(* CODESYS project PLS2 Trykkregulering 19.07.2021.ecp

Project tree, tasks and I/O mapping:
  PFCx00_SmartCoupler : 750-8212 PFC200 2ETH RS, WAGO, order no. 0750-8212, version 5.15.4.20
    application PLS2_Trykkregulering
      libraries: ; VisuDialogs, * (System); WagoTypesCommon, 1.5.3.0 (WAGO); WagoAppHART, 1.7.1.0 (WAGO); WagoAppSolenoid, 1.7.1.0 (WAGO); WagoAppPowerMeasurement, 1.7.1.0 (WAGO); WagoTypesCom, 1.6.1.2 (WAGO); WagoAppDALI, 1.3.0.33 (WAGO); WagoSysKbusModule, 1.8.2.0 (WAGO); WagoSysKbusServices, 1.8.7.4 (WAGO); WagoAppPlcModbus, 1.1.2.21 (WAGO); WagoTypesAsync_Internal_Template, 1.0.0.1 (WAGO); WagoSysModule_75x_632, 1.8.1.0 (WAGO); WagoSysModule_75x_48x, 1.5.1.0 (WAGO); WagoVisuIcons, 1.0.1.0 (WAGO); WagoSysModule_75x_49x, 1.7.1.0 (WAGO); WagoSysModule_753_647, 1.1.1.0 (WAGO); WagoAppKNX, 1.0.4.0 (WAGO); WagoAppCloud, * (WAGO); WagoAppTime, 1.7.3.3 (WAGO); WagoAppJSON, 1.0.2.0 (WAGO); CmpEventMgr, 3.5.12.0 (System); Component Manager, 3.5.13.0 (System); CmpApp, 3.5.13.0 (System); CmpIecTask, 3.5.13.0 (System)
      task PLC_Task (cyclic, interval 100 ms, priority 10, watchdog 90 ms x 1) calls PLC_PRG
      task VISU_TASK (cyclic, interval 100 ms, priority 15) calls VisuElems.Visu_Prg
      task TrendRecordingTask (cyclic, interval 100 ms, priority 15) calls VisuTrendStorageAccess.GlobalInstances.g_TrendRecordingManager.CyclicCall
      program PLC_PRG [ST]
      program Alarms [ST]
      GlobalData/
        global variables HMI
        global variables Local
        global variables IO
        global variables SIM
        global variables STATUS
      Symbols
      program Inputs [ST]
      program Control [ST]
      program Outputs [ST]
      program Simulation [ST]
      program Initialize [ST]
      visualisation Visualization
      global variables PersistentVars
      function RestartOpcUaMqttLinkOnDownload [ST]
      function RestartOpcUaMqttLinkOnOnlineChange [ST]
    ProjectConfigurationTxt
    ProjectConfiguration
    Common.PCI
    Kbus : Kbus, WAGO, version 1.4.0.2
        unmapped channels: K-BUS diagnostics
    MODBUS
      MODBUS : MODBUS, WAGO, order no. n/a, version 1.1.1.15
    Serial
      COM1 : COM1, WAGO, version 0.0.0.19
  00000000-0000-0000-0000-000000000000|C:\Users\WagoNorgeLab-1\AppData\Local\Temp\ee55296a4ebe4169b370fb7549785af2\ProjectCfg.txt
  LibFB/
    function block AlarmDigitalFB [ST]
    function block MotorDigitalFB [ST]
    function block ControlAnalogFB [ST]
    function block ScalingFB [ST]
    function block signalDigitalFB [ST]
    function block TimerFB [ST]
    function block SignalAnalogFB [ST]
    function block PIDFB [ST]
    function block WorkDistributorFB [ST]
  LibHmiStructs/
    data type AlarmDigitalHmiPv
    data type ControlAnalogHmiPv
    data type MotorDigitalHmiPv
    data type MotorDigitalHmiCmd
    data type ControlAnalogHmiCmd
    data type AlarmDigitalHmiCmd
    data type TimerHmiPv
    data type TimerHmiCmd
    data type SignalDigitalHmiPv
    data type SignalDigitalHmiCmd
    data type ScalingHmiPv
    data type ScalingHmiCmd
    data type SignalAnalogHmiPv
    data type SignalAnalogHmiCmd
    data type AliveHmiPv
    data type PIDHmiCmd
    data type PIDHmiPv
    data type WorkDistributorHmiPv
  Utils/
    function eulers [ST]
    function process [ST]
    function String_To_ForcastArray [ST]
    data type OpcUa_Mqtt_Status
    function firstOrderSystem [ST]
  text list GlobalTextList
  00000000-0000-0000-0000-000000000000|C:\Users\WagoNorgeLab-1\AppData\Local\Temp\0890fa1c76c045128ce9e2a1421b24b3\Project.xml
*)

// LibHmiStructs/AlarmDigitalHmiPv
// These are autogenerated, do not manual modify it
TYPE AlarmDigitalHmiPv :
STRUCT
	_tagId: STRING;
	_type: STRING;
	_owner: STRING;
	Input_Pv:	BOOL;
	Delay:	TimerHmiPv;
	Alarm:	BOOL;
END_STRUCT
END_TYPE

// LibHmiStructs/ControlAnalogHmiPv
// These are autogenerated, do not manual modify it
TYPE ControlAnalogHmiPv :
STRUCT
	_tagId: STRING;
	_type: STRING;
	_owner: STRING;
	ControlValue_Pv:	REAL;
	Interlocked_Pv:	BOOL;
	AlarmControlFailed:	AlarmDigitalHmiPv;
	Feedback_Pv:REAL;
	RunHours_Pv:INT;
	RunMinutes_Pv:int;
END_STRUCT
END_TYPE

// LibHmiStructs/MotorDigitalHmiPv
// These are autogenerated, do not manual modify it
TYPE MotorDigitalHmiPv :
STRUCT
_tagId: STRING;
_type: STRING;
_owner: STRING;
Interlocked_Pv:BOOL;
ControlValue_Pv:BOOL;
AlarmStartFailed:AlarmDigitalHmiPv;
AlarmStopFailed:AlarmDigitalHmiPv;
Started_Pv:BOOL;
Stopped_Pv:BOOL;
END_STRUCT
END_TYPE

// LibHmiStructs/MotorDigitalHmiCmd
// These are autogenerated, do not manual modify it
TYPE MotorDigitalHmiCmd :
STRUCT
_tagId: STRING;
_type: STRING;
_owner: STRING;
Tag:STRING;
Description:STRING;
Auto:BOOL;
AlarmStartFailed:AlarmDigitalHmiCmd;
AlarmStopFailed:AlarmDigitalHmiCmd;
ManualStart_Cmd:BOOL;
END_STRUCT
END_TYPE

// LibHmiStructs/ControlAnalogHmiCmd
// These are autogenerated, do not manual modify it
TYPE ControlAnalogHmiCmd :
STRUCT
	_tagId: STRING;
	_type: STRING;
	_owner: STRING;
	Tag:STRING;
	Description:STRING;
	Auto:BOOL;
	ManualControlValue_Cmd:REAL;
	AlarmControlFailed:	AlarmDigitalHmiCmd;
	AlarmControlFailedLimit:	REAL;
END_STRUCT
END_TYPE

// LibHmiStructs/AlarmDigitalHmiCmd
// These are autogenerated, do not manual modify it
TYPE AlarmDigitalHmiCmd :
STRUCT
	_tagId: STRING;
	_type: STRING;
	_owner: STRING;
	Tag:	STRING;
	Description:	STRING;
	Delay:	TimerHmiCmd;
	Acknowledged:	BOOL;
END_STRUCT
END_TYPE

// LibHmiStructs/TimerHmiPv
// These are autogenerated, do not manual modify it
TYPE TimerHmiPv :
STRUCT
	_tagId:STRING;
	_type: STRING;
	_owner: STRING;
	Input_Pv:	BOOL;
	Output_Pv:	BOOL;
	OnDelayElapsed:	REAL;
	OffDelayElapsed:	REAL;
END_STRUCT
END_TYPE

// LibHmiStructs/TimerHmiCmd
// These are autogenerated, do not manual modify it
TYPE TimerHmiCmd :
STRUCT
	_tagId:STRING;
	_type: STRING;
	_owner: STRING;
	Tag:	STRING;
	Description:	STRING;
	OnDelayLimit:	REAL;
	OffDelayLimit:	REAL;
END_STRUCT
END_TYPE

// LibHmiStructs/SignalDigitalHmiPv
// These are autogenerated, do not manual modify it
TYPE SignalDigitalHmiPv :
STRUCT
_tagId: STRING;
_type: STRING;
_owner: STRING;
Input_Pv:BOOL;
Output_Pv:BOOL;
END_STRUCT
END_TYPE

// LibHmiStructs/SignalDigitalHmiCmd
// These are autogenerated, do not manual modify it
TYPE SignalDigitalHmiCmd :
STRUCT
_tagId: STRING;
_type: STRING;
_owner: STRING;
Tag:STRING;
Description:STRING;
SimulationMode:BOOL;
SimulationValue:BOOL;
END_STRUCT
END_TYPE

// LibHmiStructs/ScalingHmiPv
// These are autogenerated, do not manual modify it
TYPE ScalingHmiPv :
STRUCT
_tagId: STRING;
_type: STRING;
_owner: STRING;
Input_Pv:REAL;
Output_Pv:REAL;
END_STRUCT
END_TYPE

// LibHmiStructs/ScalingHmiCmd
// These are autogenerated, do not manual modify it
TYPE ScalingHmiCmd :
STRUCT
	_tagId: STRING;
	_type: STRING;
	_owner: STRING;
	InputUnit:STRING;
	InputMin_Cmd:REAL;
	InputMax_Cmd:REAL;
	OutputUnit:STRING;
	OutputMin_Cmd:REAL;
	OutputMax_Cmd:REAL;
END_STRUCT
END_TYPE

// LibHmiStructs/SignalAnalogHmiPv
// These are autogenerated, do not manual modify it
TYPE SignalAnalogHmiPv :
STRUCT
_tagId: STRING;
_type: STRING;
_owner: STRING;
RawInput_Pv:REAL;
Output_Pv:REAL;
AlarmHigh:AlarmDigitalHmiPv;
AlarmHighHigh:AlarmDigitalHmiPv;
AlarmLow:AlarmDigitalHmiPv;
AlarmLowLow:AlarmDigitalHmiPv;
InputScaling:ScalingHmiPv;
END_STRUCT
END_TYPE

// LibHmiStructs/SignalAnalogHmiCmd
// These are autogenerated, do not manual modify it
TYPE SignalAnalogHmiCmd :
STRUCT
_tagId: STRING;
_type: STRING;
_owner: STRING;
Tag:STRING;
Description:STRING;
AlarmHigh:AlarmDigitalHmiCmd;
AlarmHighHigh:AlarmDigitalHmiCmd;
AlarmLow:AlarmDigitalHmiCmd;
AlarmLowLow:AlarmDigitalHmiCmd;
AlarmHighLimit:REAL;
AlarmHighHighLimit:REAL;
AlarmLowLimit:REAL;
AlarmLowLowLimit:REAL;
AlarmHysteresis:REAL;
SimulationMode:BOOL;
SimulationValue:REAL;
InputScaling:ScalingHmiCmd;
END_STRUCT
END_TYPE

// LibHmiStructs/AliveHmiPv
TYPE AliveHmiPv :
STRUCT
	_tagId:STRING;
	_type: STRING;
	_owner: STRING;
	CounterPv:INT;
END_STRUCT
END_TYPE

// LibHmiStructs/PIDHmiCmd
TYPE PIDHmiCmd :
STRUCT
	_tagId: STRING;
	_type: STRING;
	_owner: STRING;
	Tag:STRING;
	Description:STRING;
	K:REAL;
	EnableK:BOOL;
	Ti:REAL;
	EnableI:BOOL;
	Td:REAL;
	N:REAL;
	EnableD:BOOL;
	Auto:BOOL;
	ManualValue_Cmd:REAL;
	u0:REAL;
	TrackingGain:REAL;
	HmiReference_Cmd:REAL;
	HmiReference:BOOL;
END_STRUCT
END_TYPE

// LibHmiStructs/PIDHmiPv
TYPE PIDHmiPv :
STRUCT
	_tagId: STRING;
	_type: STRING;
	_owner: STRING;
	Reference_Pv:REAL;
	ProcessMeasure:REAL;
	Error:REAL;
	Output:REAL;
	up:REAL;
	ui:REAL;
	ud:REAL;
	es:REAL;
	u:REAL;
END_STRUCT
END_TYPE

// Utils/OpcUa_Mqtt_Status
TYPE OpcUa_Mqtt_Status :
STRUCT
	LastRun:STRING;
	AliveCounterPv:INT := 0;
	Restart_Cmd:BOOL := FALSE;
END_STRUCT
END_TYPE

// LibHmiStructs/WorkDistributorHmiPv
TYPE WorkDistributorHmiPv :
STRUCT
_tagId:STRING;
_type:STRING;
_owner:STRING;
Tag1:STRING;
Tag2:STRING;
Tag3:STRING;
RunHours1:INT;
RunHours2:INT;
RunHours3:INT;
AlarmNotAuto:BOOL;
END_STRUCT
END_TYPE

// PFCx00_SmartCoupler/PLS2_Trykkregulering/GlobalData/HMI
{attribute 'qualified_only'}
VAR_GLOBAL PERSISTENT RETAIN
AliveCounterPlc2Pv:AliveHmiPv;

DeliveryPump1Cmd:ControlAnalogHmiCmd;
DeliveryPump1Pv:ControlAnalogHmiPv;
DeliveryPump2Cmd:ControlAnalogHmiCmd;
DeliveryPump2Pv:ControlAnalogHmiPv;
DeliveryPump3Cmd:ControlAnalogHmiCmd;
DeliveryPump3Pv:ControlAnalogHmiPv;
DeliveryPumpPIDCmd:PIDHmiCmd;
DeliveryPumpPIDPv:PIDHmiPv;
DeliveryPumpWorkDistPv:WorkDistributorHmiPv;
TreatmentPressureCmd:SignalAnalogHmiCmd;
TreatmentPressurePv:SignalAnalogHmiPv;
ConsumerPressureCmd:SignalAnalogHmiCmd;
ConsumerPressurePv:SignalAnalogHmiPv;
END_VAR

// PFCx00_SmartCoupler/PLS2_Trykkregulering/GlobalData/Local
{attribute 'qualified_only'}
VAR_GLOBAL
DeliveryPump1:ControlAnalogFB;
DeliveryPump2:ControlAnalogFB;
DeliveryPump3:ControlAnalogFB;
DeliveryPumpPID:PIDFB;
DeliveryPumpWorkDist:WorkDistributorFB;
TreatmentPressure:SignalAnalogFB;
ConsumerPressure:SignalAnalogFB;
END_VAR

// PFCx00_SmartCoupler/PLS2_Trykkregulering/GlobalData/IO
{attribute 'qualified_only'}
VAR_GLOBAL
AI_DeliveryPump1SpeedPv:REAL;
AI_DeliveryPump2SpeedPv:Real;
AI_DeliveryPump3SpeedPv:Real;

AO_DeliveryPump1ControlValue:real;
AO_DeliveryPump2ControlValue:real;
AO_DeliveryPump3ControlValue:REAL;

AI_ConsumerPressurePv:REAL;
AI_TreatmentPressurePv:REAL;
END_VAR

// PFCx00_SmartCoupler/PLS2_Trykkregulering/GlobalData/SIM
{attribute 'qualified_only'}
VAR_GLOBAL
	Disturbance:REAL;
	Process_y:REAL;
	Process:REAL;
	Ref:REAL;
	Output:REAL;
END_VAR

// PFCx00_SmartCoupler/PLS2_Trykkregulering/GlobalData/STATUS
{attribute 'qualified_only'}
VAR_GLOBAL
	OpcUaMqttLinkStatus: OpcUa_Mqtt_Status;
END_VAR

// PFCx00_SmartCoupler/PLS2_Trykkregulering/PersistentVars
{attribute 'qualified_only'}
VAR_GLOBAL PERSISTENT RETAIN
	// Generated instance path of persistent variable
	HMI.AliveCounterPlc2Pv: AliveHmiPv;
	// Generated instance path of persistent variable
	HMI.DeliveryPump1Cmd: ControlAnalogHmiCmd;
	// Generated instance path of persistent variable
	HMI.DeliveryPump1Pv: ControlAnalogHmiPv;
	// Generated instance path of persistent variable
	HMI.DeliveryPump2Cmd: ControlAnalogHmiCmd;
	// Generated instance path of persistent variable
	HMI.DeliveryPump2Pv: ControlAnalogHmiPv;
	// Generated instance path of persistent variable
	HMI.DeliveryPump3Cmd: ControlAnalogHmiCmd;
	// Generated instance path of persistent variable
	HMI.DeliveryPump3Pv: ControlAnalogHmiPv;
	// Generated instance path of persistent variable
	HMI.DeliveryPumpPIDCmd: PIDHmiCmd;
	// Generated instance path of persistent variable
	HMI.DeliveryPumpPIDPv: PIDHmiPv;
	// Generated instance path of persistent variable
	HMI.DeliveryPumpWorkDistPv: WorkDistributorHmiPv;
	// Generated instance path of persistent variable
	HMI.TreatmentPressureCmd: SignalAnalogHmiCmd;
	// Generated instance path of persistent variable
	HMI.TreatmentPressurePv: SignalAnalogHmiPv;
	// Generated instance path of persistent variable
	HMI.ConsumerPressureCmd: SignalAnalogHmiCmd;
	// Generated instance path of persistent variable
	HMI.ConsumerPressurePv: SignalAnalogHmiPv;
END_VAR

// PFCx00_SmartCoupler/PLS2_Trykkregulering/PLC_PRG
PROGRAM PLC_PRG
VAR
	_firstScan:BOOL := TRUE;
	_counter:INT;
	_lastRun:STRING;
END_VAR



// Signaling that the PLC is alive
Hmi.AliveCounterPlc2Pv._tagId := 'AliveCounterPlc2Pv';
Hmi.AliveCounterPlc2Pv._type := 'AliveHmi';
Hmi.AliveCounterPlc2Pv._owner := 'plc2';
HMI.AliveCounterPlc2Pv.CounterPv := HMI.AliveCounterPlc2Pv.CounterPv + 1;

_counter := STATUS.OpcUaMqttLinkStatus.AliveCounterPv;
_lastRun := STATUS.OpcUaMqttLinkStatus.LastRun;

IF _firstScan THEN
	Initialize();
END_IF
Inputs();
Alarms();
Control();
Outputs();
Simulation();





// Always last
_firstScan := FALSE;

END_PROGRAM

// PFCx00_SmartCoupler/PLS2_Trykkregulering/Initialize
PROGRAM Initialize
VAR
END_VAR



Hmi.DeliveryPumpPIDCmd.Tag := 'PID01';
Hmi.DeliveryPumpPIDCmd.Description := 'Regulator for controling pressure';
Hmi.DeliveryPumpPIDCmd.Auto := TRUE;
Hmi.DeliveryPumpPIDCmd.EnableK := TRUE;
Hmi.DeliveryPumpPIDCmd.EnableI := TRUE;
Hmi.DeliveryPumpPIDCmd.EnableD := TRUE;
Hmi.DeliveryPumpPIDCmd.K := 8.0;
Hmi.DeliveryPumpPIDCmd.Ti := 5.5;
Hmi.DeliveryPumpPIDCmd.Td := 0.5;
Hmi.DeliveryPumpPIDCmd.N := 10.0;
Hmi.DeliveryPumpPIDCmd.TrackingGain := 1.0;
Hmi.DeliveryPumpPIDCmd.u0 := 50.0;


HMI.DeliveryPump1Cmd.Tag := 'P01';
HMI.DeliveryPump1Cmd.Description := 'Delivery pump 1';
HMI.DeliveryPump1Cmd.Auto := TRUE;
HMI.DeliveryPump1Cmd.ManualControlValue_Cmd := 50.0;
HMI.DeliveryPump1Cmd.AlarmControlFailedLimit := 10.0;
HMI.DeliveryPump1Cmd.AlarmControlFailed.Description := 'Failed to control Delivery Pump 1';
HMI.DeliveryPump1Cmd.AlarmControlFailed.Delay.OnDelayLimit := 10.0;
HMI.DeliveryPump1Cmd.AlarmControlFailed.Delay.OffDelayLimit := 10.0;
HMI.DeliveryPump1Cmd.AlarmControlFailed.Acknowledged := TRUE;

HMI.DeliveryPump2Cmd.Tag := 'P02';
HMI.DeliveryPump2Cmd.Description := 'Delivery pump 2';
HMI.DeliveryPump2Cmd.Auto := TRUE;
HMI.DeliveryPump2Cmd.ManualControlValue_Cmd := 50.0;
HMI.DeliveryPump2Cmd.AlarmControlFailedLimit := 10.0;
HMI.DeliveryPump2Cmd.AlarmControlFailed.Description := 'Failed to control Delivery Pump 2';
HMI.DeliveryPump2Cmd.AlarmControlFailed.Delay.OnDelayLimit := 10.0;
HMI.DeliveryPump2Cmd.AlarmControlFailed.Delay.OffDelayLimit := 10.0;
HMI.DeliveryPump2Cmd.AlarmControlFailed.Acknowledged := TRUE;

HMI.DeliveryPump3Cmd.Tag := 'P03';
HMI.DeliveryPump3Cmd.Description := 'Delivery pump 2';
HMI.DeliveryPump3Cmd.Auto := TRUE;
HMI.DeliveryPump3Cmd.ManualControlValue_Cmd := 50.0;
HMI.DeliveryPump3Cmd.AlarmControlFailedLimit := 10.0;
HMI.DeliveryPump3Cmd.AlarmControlFailed.Description := 'Failed to control Delivery Pump 3';
HMI.DeliveryPump3Cmd.AlarmControlFailed.Delay.OnDelayLimit := 10.0;
HMI.DeliveryPump3Cmd.AlarmControlFailed.Delay.OffDelayLimit := 10.0;
HMI.DeliveryPump3Cmd.AlarmControlFailed.Acknowledged := TRUE;

Hmi.TreatmentPressureCmd.Tag := 'PT02';
Hmi.TreatmentPressureCmd.Description := 'Treatment pressure';
Hmi.TreatmentPressureCmd.AlarmHysteresis := 3.0;
Hmi.TreatmentPressureCmd.AlarmHighHighLimit := 90.0;
Hmi.TreatmentPressureCmd.AlarmHighLimit := 80.0;
Hmi.TreatmentPressureCmd.AlarmLowLowLimit := 10.0;
Hmi.TreatmentPressureCmd.AlarmLowLimit := 20.0;
Hmi.TreatmentPressureCmd.AlarmHigh.Description := 'High Treatment Pressure';
Hmi.TreatmentPressureCmd.AlarmHighHigh.Description := 'High high Treatment Pressure';
Hmi.TreatmentPressureCmd.AlarmLow.Description := 'Low Treatment Pressure';
Hmi.TreatmentPressureCmd.AlarmLowLow.Description := 'Low low Treatment Pressure';
Hmi.TreatmentPressureCmd.AlarmHigh.Delay.OnDelayLimit := 1.0;
Hmi.TreatmentPressureCmd.AlarmHigh.Delay.OffDelayLimit := 1.0;
Hmi.TreatmentPressureCmd.AlarmHighHigh.Delay.OnDelayLimit := 1.0;
Hmi.TreatmentPressureCmd.AlarmHighHigh.Delay.OffDelayLimit := 1.0;
Hmi.TreatmentPressureCmd.AlarmLow.Delay.OnDelayLimit := 1.0;
Hmi.TreatmentPressureCmd.AlarmLow.Delay.OffDelayLimit := 1.0;
Hmi.TreatmentPressureCmd.AlarmLowLow.Delay.OnDelayLimit := 1.0;
Hmi.TreatmentPressureCmd.AlarmLowLow.Delay.OffDelayLimit := 1.0;
Hmi.TreatmentPressureCmd.InputScaling.InputUnit := 'na';
Hmi.TreatmentPressureCmd.InputScaling.OutputUnit := 'bar';
Hmi.TreatmentPressureCmd.InputScaling.InputMax_Cmd := 100.0;
Hmi.TreatmentPressureCmd.InputScaling.InputMin_Cmd := 0.0;
Hmi.TreatmentPressureCmd.InputScaling.OutputMax_Cmd := 100.0;
Hmi.TreatmentPressureCmd.InputScaling.OutputMin_Cmd := 0.0;

Hmi.ConsumerPressureCmd.Tag := 'PT03';
Hmi.ConsumerPressureCmd.Description := 'Consumer pressure';
Hmi.ConsumerPressureCmd.AlarmHysteresis := 3.0;
Hmi.ConsumerPressureCmd.AlarmHighHighLimit := 90.0;
Hmi.ConsumerPressureCmd.AlarmHighLimit := 80.0;
Hmi.ConsumerPressureCmd.AlarmLowLowLimit := 10.0;
Hmi.ConsumerPressureCmd.AlarmLowLimit := 20.0;
Hmi.ConsumerPressureCmd.AlarmHigh.Description := 'High Consumer Pressure';
Hmi.ConsumerPressureCmd.AlarmHighHigh.Description := 'High high Consumer Pressure';
Hmi.ConsumerPressureCmd.AlarmLow.Description := 'Low Consumer Pressure';
Hmi.ConsumerPressureCmd.AlarmLowLow.Description := 'Low low Consumer Pressure';
Hmi.ConsumerPressureCmd.AlarmHigh.Delay.OnDelayLimit := 1.0;
Hmi.ConsumerPressureCmd.AlarmHigh.Delay.OffDelayLimit := 1.0;
Hmi.ConsumerPressureCmd.AlarmHighHigh.Delay.OnDelayLimit := 1.0;
Hmi.ConsumerPressureCmd.AlarmHighHigh.Delay.OffDelayLimit := 1.0;
Hmi.ConsumerPressureCmd.AlarmLow.Delay.OnDelayLimit := 1.0;
Hmi.ConsumerPressureCmd.AlarmLow.Delay.OffDelayLimit := 1.0;
Hmi.ConsumerPressureCmd.AlarmLowLow.Delay.OnDelayLimit := 1.0;
Hmi.ConsumerPressureCmd.AlarmLowLow.Delay.OffDelayLimit := 1.0;
Hmi.ConsumerPressureCmd.InputScaling.InputUnit := 'na';
Hmi.ConsumerPressureCmd.InputScaling.OutputUnit := 'bar';
Hmi.ConsumerPressureCmd.InputScaling.InputMax_Cmd := 100.0;
Hmi.ConsumerPressureCmd.InputScaling.InputMin_Cmd := 0.0;
Hmi.ConsumerPressureCmd.InputScaling.OutputMax_Cmd := 100.0;
Hmi.ConsumerPressureCmd.InputScaling.OutputMin_Cmd := 0.0;

END_PROGRAM

// PFCx00_SmartCoupler/PLS2_Trykkregulering/Control
PROGRAM Control
VAR
	
END_VAR



// Regulator block
Local.DeliveryPumpPID(_id := 'DeliveryPumpPID', _owner := 'plc2',
	InputReference := 6.0,
	ProcessMeasure := IO.AI_ConsumerPressurePv,
	Ts := 0.1,
	uMax := 100.0,
	uMin := 0.0,
	HmiCmd := Hmi.DeliveryPumpPIDCmd,
	HmiPv := Hmi.DeliveryPumpPIDPv);

// Work distribution
Local.DeliveryPumpWorkDist(_id := 'DeliveryPumpWorkDist', _owner := 'plc2',
	InputControlSignal := Local.DeliveryPumpPID.Output,
	Tag1 := Hmi.DeliveryPump1Cmd.Tag,
	Tag2 := Hmi.DeliveryPump2Cmd.Tag,
	Tag3 := Hmi.DeliveryPump3Cmd.Tag,
	InAuto1 := Hmi.DeliveryPump1Cmd.Auto,
	InAuto2 := Hmi.DeliveryPump2Cmd.Auto,
	InAuto3 := Hmi.DeliveryPump3Cmd.Auto,
	RunHours1 := Hmi.DeliveryPump1Pv.RunHours_Pv,
	RunHours2 := Hmi.DeliveryPump2Pv.RunHours_Pv,
	RunHours3 := Hmi.DeliveryPump3Pv.RunHours_Pv,
	ChangeInterval := 60.0,
	HmiPv := HMI.DeliveryPumpWorkDistPv);
	

// Pumps
Local.DeliveryPump1(_id := 'DeliveryPump1', _owner := 'plc2',
	HmiCmd := HMI.DeliveryPump1Cmd,
	HmiPv := HMI.DeliveryPump1Pv,
	Interlock := FALSE,
	Feedback := IO.AI_DeliveryPump1SpeedPv,
	ControlValueAuto_Cmd := Local.DeliveryPumpWorkDist.Out1);
	
Local.DeliveryPump2(_id := 'DeliveryPump2', _owner := 'plc2',
	HmiCmd := HMI.DeliveryPump2Cmd,
	HmiPv := HMI.DeliveryPump2Pv,
	Interlock := FALSE,
	Feedback := IO.AI_DeliveryPump2SpeedPv,
	ControlValueAuto_Cmd := Local.DeliveryPumpWorkDist.Out2);

Local.DeliveryPump3(_id := 'DeliveryPump3', _owner := 'plc2',
	HmiCmd := HMI.DeliveryPump3Cmd,
	HmiPv := HMI.DeliveryPump3Pv,
	Interlock := FALSE,
	Feedback := IO.AI_DeliveryPump3SpeedPv,
	ControlValueAuto_Cmd := Local.DeliveryPumpWorkDist.Out3);

END_PROGRAM

// PFCx00_SmartCoupler/PLS2_Trykkregulering/Inputs
PROGRAM Inputs
VAR
	
END_VAR


				
Local.TreatmentPressure(_id := 'TreatmentPressure', _owner := 'plc2',
				RawInput := IO.AI_TreatmentPressurePv,
				HmiCmd := HMI.TreatmentPressureCmd,
				HmiPv := HMI.TreatmentPressurePv);

Local.ConsumerPressure(_id := 'ConsumerPressure', _owner := 'plc2',
				RawInput := IO.AI_ConsumerPressurePv,
				HmiCmd := HMI.ConsumerPressureCmd,
				HmiPv := HMI.ConsumerPressurePv);

END_PROGRAM

// PFCx00_SmartCoupler/PLS2_Trykkregulering/Alarms
PROGRAM Alarms
VAR
END_VAR

END_PROGRAM

// PFCx00_SmartCoupler/PLS2_Trykkregulering/Outputs
PROGRAM Outputs
VAR
END_VAR



IO.AO_DeliveryPump1ControlValue := Local.DeliveryPump1.ControlValue;
IO.AO_DeliveryPump2ControlValue := Local.DeliveryPump2.ControlValue;
IO.AO_DeliveryPump3ControlValue := Local.DeliveryPump3.ControlValue;

END_PROGRAM

// PFCx00_SmartCoupler/PLS2_Trykkregulering/Simulation
PROGRAM Simulation
VAR
	_simDelay: ARRAY[0..20] OF REAL;
	_iprocess:INT := 13; // Endret fra 19 til 13. -Peder
	_idelay:INT := 0;
	pressureDisturbance: ARRAY[0..29] OF REAL := [ 0.9,
            0.9,
            0.85,
            0.85,
			0.8,
            0.8,
            0.75,
            0.75,
            0.7,
			0.75,
            0.75,
            0.8,
            0.8,
            0.85,
			0.85,
            0.9,
            0.9,
            0.95,
            0.95,
			1.0,
            1.0,
            1.05,
            1.05,
            1.1,
			1.1,
            1.05,
            1.05,
            1.0,
            0.95,
			0.9];
			timeNow: TIME;
			secondsNow:LWORD;
			fakeHour:LWORD;
			currentFakeHour:LWORD;
END_VAR

IO.AI_DeliveryPump1SpeedPv := IO.AO_DeliveryPump1ControlValue;
IO.AI_DeliveryPump2SpeedPv := IO.AO_DeliveryPump2ControlValue;
IO.AI_DeliveryPump3SpeedPv := IO.AO_DeliveryPump3ControlValue;

timeNow := TIME();
secondsNow := (TIME_TO_LWORD(timeNow)/1000) MOD 60;
fakeHour := secondsNow/2;
SIM.Disturbance := pressureDisturbance[fakeHour];
Sim.Output := Local.DeliveryPumpPID.Output;
Sim.Ref := HMI.DeliveryPumpPIDPv.Reference_Pv;

SIM.Process_y := process(u := _simDelay[_idelay MOD 19],
	Ts := 0.1, y := SIM.Process_Y, yMin := 0, yMax := 8.0, T :=5,  Kp := 1.0);
_idelay := _idelay + 1;

_simDelay[_iprocess MOD 19] :=((IO.AI_DeliveryPump1SpeedPv + IO.AI_DeliveryPump2SpeedPv + IO.AI_DeliveryPump3SpeedPv)/10);
_iprocess := _iprocess + 1;


SIM.Process:=SIM.Process_y-SIM.Disturbance;

IO.AI_ConsumerPressurePv := SIM.Process; 
IO.AI_TreatmentPressurePv := 5.0;

END_PROGRAM

// Utils/process
FUNCTION process : REAL
VAR_INPUT
	u:REAL;
	Ts:REAL;
	y:REAL;
	yMin:REAL;
	yMax:REAL;
	T:REAL;
	Kp:REAL;
END_VAR
VAR
	_out:real;
END_VAR

_out := eulers(y, firstOrderSystem(T, Kp, y, u), Ts);
IF _out > yMax THEN
	_out := yMax;
ELSIF _out < yMin THEN
	_out := yMin;
END_IF;
process := _out;

END_FUNCTION

// Utils/eulers
FUNCTION eulers : REAL
VAR_INPUT
	y:REAL;
	f:REAL;
	h:REAL;
END_VAR
VAR
END_VAR

eulers := y + (h*f);

END_FUNCTION

// Utils/firstOrderSystem
FUNCTION firstOrderSystem : REAL
VAR_INPUT
	T:REAL;
	Kp:REAL;
	y:REAL;
	u:REAL;
END_VAR
VAR
END_VAR

firstOrderSystem :=  -(y/T) + ((Kp/T)*u);

END_FUNCTION

// LibFB/AlarmDigitalFB
FUNCTION_BLOCK AlarmDigitalFB
VAR_INPUT
	_id:STRING;
	_owner:STRING;
	Input:	BOOL;
END_VAR
VAR_OUTPUT
	Alarm:	BOOL;
END_VAR
VAR
	_Delay:	TimerFB;
	_AlarmLastScan:BOOL;
	_type:string := 'AlarmDigital';
END_VAR
VAR_IN_OUT
	HmiCmd:	AlarmDigitalHmiCmd;
	HmiPv:	AlarmDigitalHmiPv;
END_VAR

(*
Name: AlarmDigitalFB
Author: Jone Vassbø
Version: 0.3
Date: 09.03.2020
Description:
- Function block for a digital alarm, with commands from HMI in seperate struct
*)

// In routine - start -
// Validate input
// In routine - end -
// Alarm routine - start
// Alarm routine - end -

// Control routine - start -
_Delay(_id := _id, _owner := _owner, Input := Input, Output => Alarm, HmiCmd := HmiCmd.Delay, HmiPv := HmiPv.Delay);
IF Alarm AND NOT _AlarmLastScan THEN // Flank
	HmiCmd.Acknowledged := FALSE;
END_IF
_AlarmLastScan := Alarm;
// Control routine - end -

// Out routine - start - 
HmiPv.Input_Pv := Input;
HmiPv.Alarm := Alarm OR NOT HmiCmd.Acknowledged;
HmiCmd._tagId := CONCAT(_id, 'Cmd');
HmiPv._tagId := CONCAT(_id, 'Pv');
HmiPv._type := _type;
HmiCmd._type := _type;
HmiPv._owner := _owner;
HmiCmd._owner := _owner;
// Out routine - end -

END_FUNCTION_BLOCK

// LibFB/TimerFB
FUNCTION_BLOCK TimerFB
VAR_INPUT
	_id:STRING;
	_owner:STRING;
	Input:	BOOL;
END_VAR
VAR_OUTPUT
	Output:	BOOL;
END_VAR
VAR
	OnDelay: TON;
	OffDelay: TOF;
	ToSec:REAL := 1000.0;
	_type:string := 'Timer';
END_VAR
VAR_IN_OUT
	HmiCmd:	TimerHmiCmd;
	HmiPv: TimerHmiPv;
END_VAR

(*
Name: TimerFB
Author: Jone Vassbø
Version: 0.4
Date: 09.03.2020
Description:
- Function block operating as a Timer with both on and off delay
*)

// In routine - start -
// Validate input
IF HmiCmd.OnDelayLimit < 0 THEN
	HmiCmd.OnDelayLimit := 0.0;
END_IF
IF HmiCmd.OffDelayLimit < 0 THEN
	HmiCmd.OnDelayLimit := 0.0;
END_IF
// In routine - end -
// Alarm routine - start
// Alarm routine - end -
// Control routine - start -
OnDelay(IN := Input,
	PT := TO_TIME(HmiCmd.OnDelayLimit*ToSec));
HmiPv.OnDelayElapsed := TO_REAL(OnDelay.ET)/ToSec;

OffDelay(IN := OnDelay.Q,
	PT := TO_TIME(HmiCmd.OffDelayLimit*ToSec));
HmiPv.OffDelayElapsed := TO_REAL(OffDelay.ET)/ToSec;

IF OnDelay.Q THEN
	Output := TRUE;
END_IF
IF NOT OffDelay.Q THEN
	Output := FALSE;
END_IF
// Control routine - end -

// Out routine - start - 
HmiPv.Input_Pv := Input;
HmiPv.Output_Pv := Output;
HmiCmd._tagId := CONCAT(_id, 'Cmd');
HmiPv._tagId := CONCAT(_id, 'Pv');
HmiPv._type := _type;
HmiCmd._type := _type;
HmiPv._owner := _owner;
HmiCmd._owner := _owner;
// Out routine - end -

END_FUNCTION_BLOCK

// LibFB/MotorDigitalFB
FUNCTION_BLOCK MotorDigitalFB
VAR_INPUT
	_id:STRING;
	_owner:STRING;
	Interlock:BOOL;
	ControlValueAuto_Cmd:BOOL;
	Started:BOOL;
	Stopped:BOOL;
END_VAR
VAR_OUTPUT
	ControlValue:BOOL;
	Alarm:BOOL;
END_VAR
VAR
	_StartFailed:AlarmDigitalFB;
	_StopFailed:AlarmDigitalFB;
	_type:string := 'MotorDigital';
END_VAR
VAR_IN_OUT
	HmiCmd:MotorDigitalHmiCmd;
	HmiPv:MotorDigitalHmiPv;
END_VAR

(*
Name: MotorDigitalFB
Author: Jone Vassbø
Version: 0.3
Date: 09.03.2020
Description:
- Function block to control a digital motor, with commands from HMI in seperate struct
*)

// In routine - start -
// Validate input
// In routine - end -
// Alarm routine - start
_StartFailed(_id := _id, _owner := _owner, Input := (NOT Started AND ControlValue) OR (Started AND NOT ControlValue),
	HmiCmd := HmiCmd.AlarmStartFailed, HmiPv := HmiPv.AlarmStartFailed);
_StopFailed(_id := _id, _owner := _owner, Input := (Stopped AND ControlValue) OR (NOT Stopped AND NOT ControlValue),
	HmiCmd := HmiCmd.AlarmStopFailed, HmiPv := HmiPv.AlarmStopFailed);
// Alarm routine - end -

// Control routine - start -
IF Interlock OR Alarm THEN
	HmiCmd.auto := FALSE;
	HmiCmd.ManualStart_Cmd := FALSE;
END_IF

IF HmiCmd.auto THEN
	ControlValue := ControlValueAuto_Cmd;
ELSE
	ControlValue := HmiCmd.ManualStart_Cmd;
END_IF
// Control routine - end -

// Out routine - start - 
Alarm := _StartFailed.Alarm OR NOT HmiCmd.AlarmStartFailed.Acknowledged OR _StopFailed.Alarm OR NOT HmiCmd.AlarmStopFailed.Acknowledged;
HmiPv.ControlValue_Pv := ControlValue;
HmiPv.Interlocked_Pv := Interlock;
HmiPv.Started_Pv := Started;
HmiPv.Stopped_Pv := Stopped;
HmiCmd._tagId := CONCAT(_id, 'Cmd');
HmiPv._tagId := CONCAT(_id, 'Pv');
HmiPv._type := _type;
HmiCmd._type := _type;
HmiPv._owner := _owner;
HmiCmd._owner := _owner;
// Out routine - end -

END_FUNCTION_BLOCK

// LibFB/ControlAnalogFB
FUNCTION_BLOCK ControlAnalogFB
VAR_INPUT
	_id:STRING;
	_owner:STRING;
	ControlValueAuto_Cmd:REAL;
	Interlock:BOOL;
	Feedback:REAL;
END_VAR
VAR_OUTPUT
	ControlValue:REAL;
	Alarm:BOOL;
END_VAR
VAR
	_AlarmControlFailed: AlarmDigitalFB;
	_hoursTimer:TON;
	_type:STRING := 'ControlAnalog';
END_VAR
VAR_IN_OUT
	HmiCmd:	ControlAnalogHmiCmd;
	HmiPv:	ControlAnalogHmiPv;
END_VAR

(*
Name: ValveAnalogFB
Author: Jone Vassbø
Version: 0.3
Date: 09.03.2020
Description:
- Function block to control a analog valve, with commands from HMI in seperate struct
*)

// In routine - start -
// Validate input
IF HmiCmd.ManualControlValue_Cmd > 100.0 THEN
	HmiCmd.ManualControlValue_Cmd := 100.0;
END_IF
IF HmiCmd.ManualControlValue_Cmd < 0.0 THEN
	HmiCmd.ManualControlValue_Cmd := 0.0;
END_IF
IF ControlValueAuto_Cmd > 100.0 THEN
	ControlValueAuto_Cmd := 100.0;
END_IF
IF ControlValueAuto_Cmd < 0.0 THEN
	ControlValueAuto_Cmd := 0.0;
END_IF
// In routine - end -
// Alarm routine - start
_AlarmControlFailed(_id := _id, _owner := _owner, Input := ABS(Feedback - ControlValue) > HmiCmd.AlarmControlFailedLimit,
	HmiCmd := HmiCmd.AlarmControlFailed, HmiPv := HmiPv.AlarmControlFailed);
// Alarm routine - end -

// Control routine - start -
IF Interlock OR Alarm THEN
	HmiCmd.Auto := FALSE;
	HmiCmd.ManualControlValue_Cmd := 0.0;
END_IF

IF HmiCmd.auto THEN
	ControlValue := ControlValueAuto_Cmd;
ELSE
	ControlValue := HmiCmd.ManualControlValue_Cmd;
END_IF

_hoursTimer(In:= (ControlValue > 0.3) AND NOT _hoursTimer.Q, PT:= T#0.0416666667S);
// Using HmiPv because the tag is retain
IF _hoursTimer.Q THEN
	HmiPv.RunMinutes_Pv := HmiPv.RunMinutes_Pv + 1; 
END_IF
IF HmiPv.RunMinutes_Pv = 60 THEN
	HmiPv.RunHours_Pv := HmiPv.RunHours_Pv + 1;
	HmiPv.RunMinutes_Pv := 0;
END_IF
IF HmiPv.RunHours_Pv < 0 THEN
	HmiPv.RunHours_Pv := 0;
END_IF

// Control routine - end -

// Out routine - start - 
Alarm := _AlarmControlFailed.Alarm OR NOT HmiCmd.AlarmControlFailed.Acknowledged;
HmiPv.ControlValue_Pv := ControlValue;
HmiPv.Interlocked_Pv := Interlock;
HmiPv.Feedback_Pv := Feedback;
HmiCmd._tagId := CONCAT(_id, 'Cmd');
HmiPv._tagId := CONCAT(_id, 'Pv');
HmiPv._type := _type;
HmiCmd._type := _type;
HmiPv._owner := _owner;
HmiCmd._owner := _owner;
// Out routine - end -

END_FUNCTION_BLOCK

// LibFB/ScalingFB
FUNCTION_BLOCK ScalingFB
VAR_INPUT
	_id:STRING;
	_owner:STRING;
	Input:REAL;
END_VAR
VAR_OUTPUT
	Output:REAL;
END_VAR
VAR
	_type:string := 'Scaling';
END_VAR
VAR_IN_OUT
	HmiCmd:ScalingHmiCmd;
	HmiPv:ScalingHmiPv;
END_VAR


(*
Name: ScalingFB
Author: Jone Vassbø
Version: 0.3
Date: 09.03.2020
Description:
- Function block for a scaling analog value, with commands from HMI in seperate struct
*)

// Control routine - start -
Output :=  HmiCmd.OutputMin_Cmd * (1 - ((Input - HmiCmd.InputMin_Cmd) / (HmiCmd.InputMax_Cmd - HmiCmd.InputMin_Cmd))) + HmiCmd.OutputMax_Cmd * ((Input - HmiCmd.InputMin_Cmd) / (HmiCmd.InputMax_Cmd - HmiCmd.InputMin_Cmd));
// Control routine - end -

// Out routine - start - 
HmiPv.Input_Pv := Input;
HmiPv.Output_Pv := Output;
HmiCmd._tagId := CONCAT(_id, 'Cmd');
HmiPv._tagId := CONCAT(_id, 'Pv');
HmiPv._type := _type;
HmiCmd._type := _type;
HmiCmd._owner := _owner;
HmiPv._owner := _owner;
// Out routine - end -

END_FUNCTION_BLOCK

// LibFB/signalDigitalFB
FUNCTION_BLOCK signalDigitalFB
VAR_INPUT
	_id:STRING;
	_owner:STRING;
	Input:BOOL;
END_VAR
VAR_OUTPUT
	Output:BOOL;
END_VAR
VAR
	_type:string := 'SignalDigital';
END_VAR
VAR_IN_OUT
	HmiCmd:SignalDigitalHmiCmd;
	HmiPv:SignalDigitalHmiPv;
END_VAR

(*
Name: signalDigitalFB
Author: Jone Vassbø
Version: 0.3
Date: 09.03.2020
Description:
- Function block for a digital signal, with commands from HMI in seperate struct
*)

// In routine - start -
// Validate input
// In routine - end -
// Alarm routine - start
// Alarm routine - end -

// Control routine - start -
IF HmiCmd.SimulationMode THEN
	Output := HmiCmd.SimulationValue;
ELSE
	Output := Input;
END_IF
// Control routine - end -

// Out routine - start - 
HmiPv.Input_Pv := Input;
HmiPv.Output_Pv := Output;
HmiCmd._tagId := CONCAT(_id, 'Cmd');
HmiPv._tagId := CONCAT(_id, 'Pv');
HmiPv._type := _type;
HmiCmd._type := _type;
HmiPv._owner := _owner;
HmiCmd._owner := _owner;
// Out routine - end -

END_FUNCTION_BLOCK

// LibFB/SignalAnalogFB
FUNCTION_BLOCK SignalAnalogFB
VAR_INPUT
	_id:STRING;
	_owner:STRING;
	RawInput:REAL;
END_VAR
VAR_OUTPUT
	Output:REAL;
	AlarmHigh:BOOL;
	AlarmHighHigh:BOOL;
	AlarmLow:BOOL;
	AlarmLowLow:BOOL;
END_VAR
VAR
	_AlarmHigh: AlarmDigitalFB;
	_AlarmHighHigh: AlarmDigitalFB;
	_AlarmLow: AlarmDigitalFB;
	_AlarmLowLow: AlarmDigitalFB;
	_Scaling: ScalingFB;
	
	_High:BOOL;
	_HighHigh:BOOL;
	_Low:BOOL;
	_LowLow:BOOL;
	
	_type:string := 'SignalAnalog';
END_VAR
VAR_IN_OUT
	HmiCmd:SignalAnalogHmiCmd;
	HmiPv:SignalAnalogHmiPv;
END_VAR

(*
Name: SignalAnalogFB
Author: Jone Vassbø
Version: 0.3
Date: 09.03.2020
Description:
- Function block for a analog signal, with alarms and commands from HMI in seperate struct
*)

// In routine - start -
// Validate input
_Scaling(_id := _id, _owner := _owner, Input:= RawInput, HmiCmd := HmiCmd.InputScaling, HmiPv := HmiPv.InputScaling);
IF HmiCmd.SimulationMode THEN
	Output := HmiCmd.SimulationValue;
ELSE
	Output := _Scaling.Output;
END_IF
// In routine - end -
// Alarm routine - start
IF Output > HmiCmd.AlarmHighLimit THEN
	_High := TRUE;
END_IF
IF Output < (HmiCmd.AlarmHighLimit - HmiCmd.AlarmHysteresis) THEN
	_High := FALSE;
END_IF
_AlarmHigh(_id := _id, _owner := _owner, Input :=  _High,
	HmiCmd := HmiCmd.AlarmHigh, HmiPv := HmiPv.AlarmHigh);

IF Output > HmiCmd.AlarmHighHighLimit THEN
	_HighHigh := TRUE;
END_IF
IF Output < (HmiCmd.AlarmHighHighLimit - HmiCmd.AlarmHysteresis) THEN
	_HighHigh := FALSE;
END_IF
_AlarmHighHigh(_id := _id, _owner := _owner, Input :=  _HighHigh,
	HmiCmd := HmiCmd.AlarmHighHigh, HmiPv := HmiPv.AlarmHighHigh);

IF Output < HmiCmd.AlarmLowLimit THEN
	_Low := TRUE;
END_IF
IF Output > (HmiCmd.AlarmLowLimit + HmiCmd.AlarmHysteresis) THEN
	_Low := FALSE;
END_IF
_AlarmLow(_id := _id, _owner := _owner, Input :=  _Low,
	HmiCmd := HmiCmd.AlarmLow, HmiPv := HmiPv.AlarmLow);
	
IF Output < HmiCmd.AlarmLowLowLimit THEN
	_LowLow := TRUE;
END_IF
IF Output > (HmiCmd.AlarmLowLowLimit + HmiCmd.AlarmHysteresis) THEN
	_LowLow := FALSE;
END_IF
_AlarmLowLow(_id := _id, _owner := _owner, Input :=  _LowLow,
	HmiCmd := HmiCmd.AlarmLowLow, HmiPv := HmiPv.AlarmLowLow);
// Alarm routine - end -

// Control routine - start -

// Control routine - end -

// Out routine - start - 
AlarmHigh := _AlarmHigh.Alarm OR NOT HmiCmd.AlarmHigh.Acknowledged;
AlarmHighHigh := _AlarmHighHigh.Alarm OR NOT HmiCmd.AlarmHighHigh.Acknowledged;
AlarmLow := _AlarmLow.Alarm OR NOT HmiCmd.AlarmLow.Acknowledged;
AlarmLowLow := _AlarmLowLow.Alarm OR NOT HmiCmd.AlarmLowLow.Acknowledged;

HmiPv.Output_Pv := Output;
HmiPv.RawInput_Pv := RawInput;
HmiCmd._tagId := CONCAT(_id, 'Cmd');
HmiPv._tagId := CONCAT(_id, 'Pv');
HmiPv._type := _type;
HmiCmd._type := _type;
HmiPv._owner := _owner;
HmiCmd._owner := _owner;
// Out routine - end -

END_FUNCTION_BLOCK

// LibFB/PIDFB
FUNCTION_BLOCK PIDFB
VAR_INPUT
	_id:STRING;
	_owner:STRING;
	InputReference:REAL;
	ProcessMeasure:REAL;
	Ts:REAL;
	uMax:REAL;
	uMin:REAL;
END_VAR
VAR_OUTPUT
	Output:REAL;
	Out_e:REAL;
	Out_up:REAL;
	Out_ui:REAL;
	Out_ud:REAL;
	Out_es:REAL;
	Out_u:REAL;
END_VAR
VAR
	_type:STRING := 'PID';
	
	y_last:REAL := 0.0;
	u_limited:REAL := 0.0;
	u:REAL := 0.0;
	e:REAL := 0.0;
	es:REAL := 0.0;
	manual_last:BOOL := FALSE;
	// P
	up:REAL := 0.0;
	// I
	alfa:REAL := 0.0;
	ui:REAL := 0.0;
	ui_last:REAL := 0.0;
	enableI_last:BOOL := TRUE;
	// D
	ud:REAL := 0.0;
	ud_last:REAL := 0.0;
	beta:REAL := 0.0;
	ref:REAL:= 0;
END_VAR
VAR_IN_OUT
	HmiCmd:PIDHmiCmd;
	HmiPv:PIDHmiPv;
END_VAR


IF HmiCmd.HmiReference THEN
	ref := HmiCmd.HmiReference_Cmd;
ELSE
	ref := InputReference;
END_IF


e := ref - ProcessMeasure;
// K
up := (HmiCmd.K * e)*BOOL_TO_REAL(HmiCmd.EnableK);

// I
alfa := Ts / HmiCmd.Ti;
ui := (ui_last + (HmiCmd.K * alfa * e) + (es*(1/HmiCmd.TrackingGain)))*BOOL_TO_REAL(HmiCmd.EnableI);        
ui_last := ui;
// On enable I
IF HmiCmd.EnableI AND NOT enableI_last THEN
	ui := HmiCmd.u0;
END_IF;
// On disable I
IF NOT HmiCmd.EnableI AND enableI_last THEN
	HmiCmd.u0 := ui;
END_IF;

enableI_last := HmiCmd.enableI;
// D
beta := HmiCmd.Td / (HmiCmd.Td + (Ts * HmiCmd.N));
ud := ((beta * ud_last) - (HmiCmd.K * (HmiCmd.Td / Ts) * (1 - beta) * (ProcessMeasure - y_last))) * BOOL_TO_REAL(HmiCmd.enableD);
ud_last := ud;
y_last := ProcessMeasure;

u := HmiCmd.u0 + up + ui + ud;

// On enable manual
IF NOT HmiCmd.Auto AND NOT manual_last THEN
	HmiCmd.ManualValue_Cmd := u;
END_IF;
IF NOT HmiCmd.Auto THEN
	u_limited := HmiCmd.ManualValue_Cmd;
ELSE
	u_limited := u;
END_IF;
IF u_limited > uMax THEN
	u_limited := uMax;
ELSIF u_limited < uMin THEN
	u_limited := uMin;
END_IF;

manual_last := NOT HmiCmd.Auto;
es := u_limited - u;

Output := u_limited;
Out_e := e;
Out_up := up;
Out_ui := ui;
Out_ud := ud;
Out_es := es;
Out_u := u;

HmiPv.Reference_Pv := ref;
HmiPv.ProcessMeasure := ProcessMeasure;
HmiPv.Error := e;
HmiPv.Output := Output;
HmiPv.up := up;
HmiPv.ui := ui;
HmiPv.ud := ud;
HmiPv.es := es;
HmiPv.u := u;

HmiCmd._tagId := CONCAT(_id, 'Cmd');
HmiPv._tagId := CONCAT(_id, 'Pv');
HmiPv._type := _type;
HmiCmd._type := _type;
HmiPv._owner := _owner;
HmiCmd._owner := _owner;

END_FUNCTION_BLOCK

// Utils/String_To_ForcastArray
FUNCTION String_To_ForcastArray : ARRAY[0..4] OF REAL
VAR_INPUT
	InputString:STRING;
END_VAR
VAR
	temp:STRING;
	temp1:STRING;
	temp2:STRING;
	pos:INT;
	i:INT;
	values :ARRAY[0..4] OF REAL;
END_VAR

i := 0;

pos := LEN(InputString);
temp := DELETE(InputString, 1, 1);
temp1 := temp;
temp := DELETE(temp, 1, pos-1);
temp2 := temp;
pos := FIND(temp, ',');
FOR i := 0 TO 3 BY 1 DO
	values[i] := STRING_TO_REAL(LEFT(temp, pos-1)); // Denne tar ikke hensyn til siste verdi, då den leter etter komma men det finnes ikke
	temp := DELETE(temp, pos+2, 0);
	pos := FIND(temp, ',');
END_FOR;
values[4] := STRING_TO_REAL(temp);
String_To_ForcastArray := values;

END_FUNCTION

// LibFB/WorkDistributorFB
FUNCTION_BLOCK WorkDistributorFB
VAR_INPUT
	_id:STRING;
	_owner:STRING;
	InputControlSignal:REAL;
	Tag1:STRING;
	Tag2:STRING;
	Tag3:STRING;
	InAuto1:BOOL;
	InAuto2:BOOL;
	InAuto3:BOOL;
	RunHours1:INT;
	RunHours2:INT;
	RunHours3:INT;
	ChangeInterval:REAL;
END_VAR
VAR_OUTPUT
	Out1:REAL;
	Out2:REAL;
	Out3:REAL;

END_VAR
VAR
	_intervalTimer:TON;
	_alarm:BOOL;
	_type:STRING := 'WorkDistributor';
	_ToSec:REAL := 1000.0;
	_maxWorkingHours:INT;
	_run1:BOOL;
	_run2:BOOL;
	_run3:BOOL;
END_VAR
VAR_IN_OUT
	HmiPv:WorkDistributorHmiPv;
END_VAR


_intervalTimer(IN := NOT _intervalTimer.Q,
	PT := TO_TIME(ChangeInterval*_ToSec));

_alarm := NOT InAuto1 OR NOT InAuto2 OR NOT InAuto3;

// These are located here because of the return statments
HmiPv.Tag1 := Tag1;
HmiPv.Tag2 := Tag2;
HmiPv.Tag3 := Tag3;
HmiPv.RunHours1 := RunHours1;
HmiPv.RunHours2 := RunHours2;
HmiPv.RunHours3 := RunHours3;
HmiPv.AlarmNotAuto := _alarm;

HmiPv._tagId := CONCAT(_id, 'Pv');
HmiPv._type := _type;
HmiPv._owner := _owner;

IF _alarm THEN
	Out1 := InputControlSignal;
	Out2 := InputControlSignal;
	Out3 := InputControlSignal;
	RETURN;
END_IF

Out1 := (InputControlSignal*BOOL_TO_REAL(_run1)); 
Out2 := (InputControlSignal*BOOL_TO_REAL(_run2));
Out3 := (InputControlSignal*BOOL_TO_REAL(_run3));


// Time to change who is working
IF _intervalTimer.Q THEN
	_run1 := TRUE;
	_run2 := TRUE;
	_run3 := TRUE;
	
	_maxWorkingHours := RunHours1;
	IF RunHours2 > _maxWorkingHours THEN
		_maxWorkingHours := RunHours2;
	END_IF
	IF RunHours3 > _maxWorkingHours THEN
		_maxWorkingHours := RunHours3;
	END_IF

	IF RunHours1 = _maxWorkingHours THEN
		_run1 := FALSE;
		RETURN; // Prevents two from stopping
	END_IF
	IF RunHours2 = _maxWorkingHours THEN
		_run2 := FALSE;
		RETURN;
	END_IF
	IF RunHours3 = _maxWorkingHours THEN
		_run3 := FALSE;
		RETURN;
	END_IF
END_IF

END_FUNCTION_BLOCK

// PFCx00_SmartCoupler/PLS2_Trykkregulering/RestartOpcUaMqttLinkOnDownload
FUNCTION RestartOpcUaMqttLinkOnDownload : DWORD
VAR_IN_OUT
	EventPrm: CmpApp.EVTPARAM_CmpApp;
END_VAR
VAR
END_VAR

(*
This function is called whan a download is about to happen. 
This will force the Opc Ua - MQTT link to restart.
The restart will take 10 seconds, allowing e!Cockpit to download and start before the link starts.
*)
Status.OpcUaMqttLinkStatus.Restart_Cmd := TRUE;

END_FUNCTION

// PFCx00_SmartCoupler/PLS2_Trykkregulering/RestartOpcUaMqttLinkOnOnlineChange
FUNCTION RestartOpcUaMqttLinkOnOnlineChange : DWORD
VAR_IN_OUT
	EventPrm: CmpApp.EVTPARAM_CmpApp;
END_VAR
VAR
END_VAR

(*
This function is called whan a online change is about to happen. 
This will force the Opc Ua - MQTT link to restart.
The restart will take 10 seconds, allowing e!Cockpit to download and start before the link starts.
*)
Status.OpcUaMqttLinkStatus.Restart_Cmd := TRUE;

END_FUNCTION

// PFCx00_SmartCoupler/PLS2_Trykkregulering/Visualization
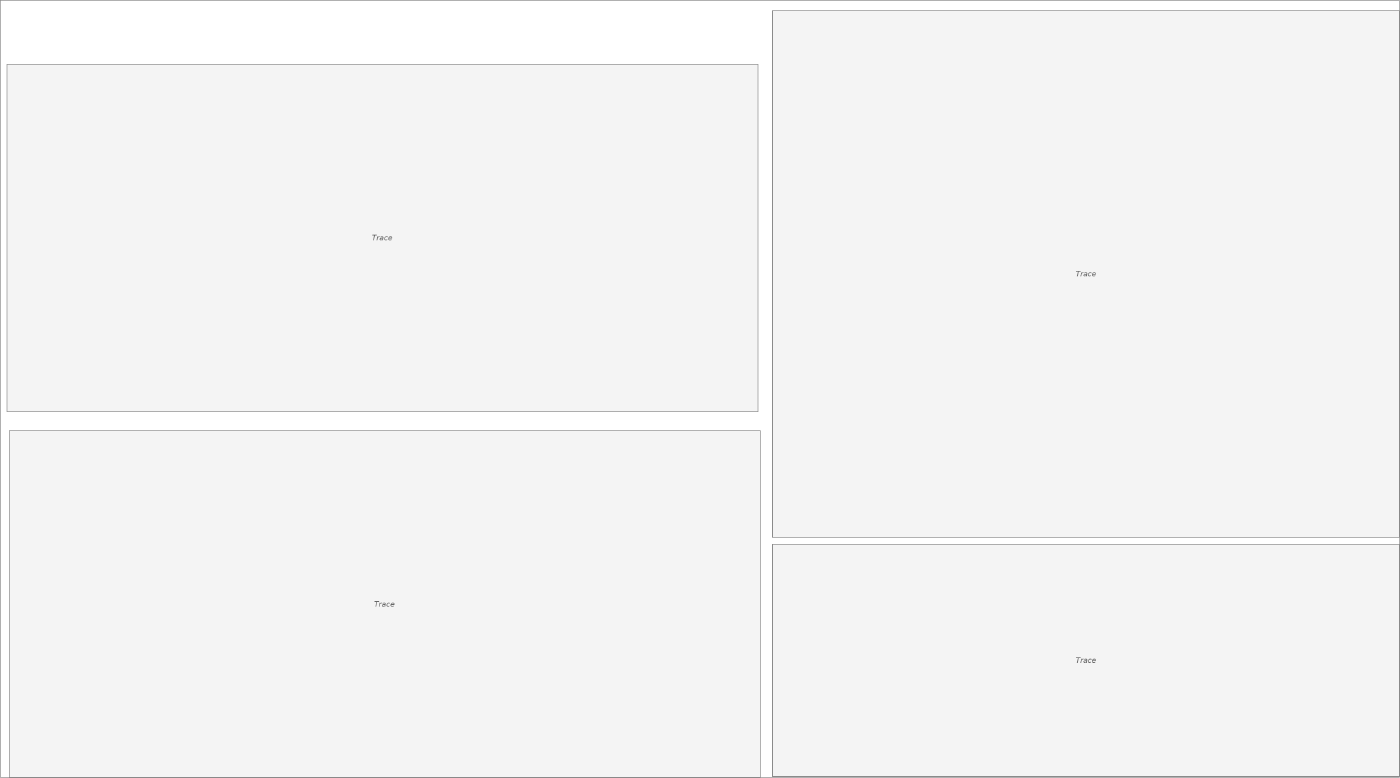
VISUALIZATION Visualization  // 1882x1047
    Trace (12,579 1010x468)
    Trace (1038,14 844x709)
    Trace (1038,732 844x313)
    Trace (9,86 1010x468)
END_VISUALIZATION
